{attribute 'qualified_only'}
{attribute 'strict'}

//-----------------------------------------------------------------------------------------
//
//                  				ENUM_Jog_Direction
//
//						Enumération des Direction des Axes en Jog			
//-----------------------------------------------------------------------------------------
//
//Auteur: G.GOETZ
//Création: 19.01.2026
//Dernière modification : 19.01.2026 (G.GOETZ)
//       			
//-----------------------------------------------------------------------------------------
//
//     							Liste des modifications  	
//
// 19.01.2026 (G.GOETZ) -> Création		
//-----------------------------------------------------------------------------------------

TYPE ENUM_Jog_Direction :
(
	None := 0 , // Unknow Direction
	Plus := 1 , // Positive Direction
	Minus := 2 // Negative Direction
);
END_TYPE

(* stored: Version 1.1.0.1, ProductVersion 3.1.4024.13
   DUT ENUM_Jog_Direction: Id {f0199e3f-95af-49c3-b1fc-b2bcf4c9c905} *)
